RoboDK station: simulator.rdk

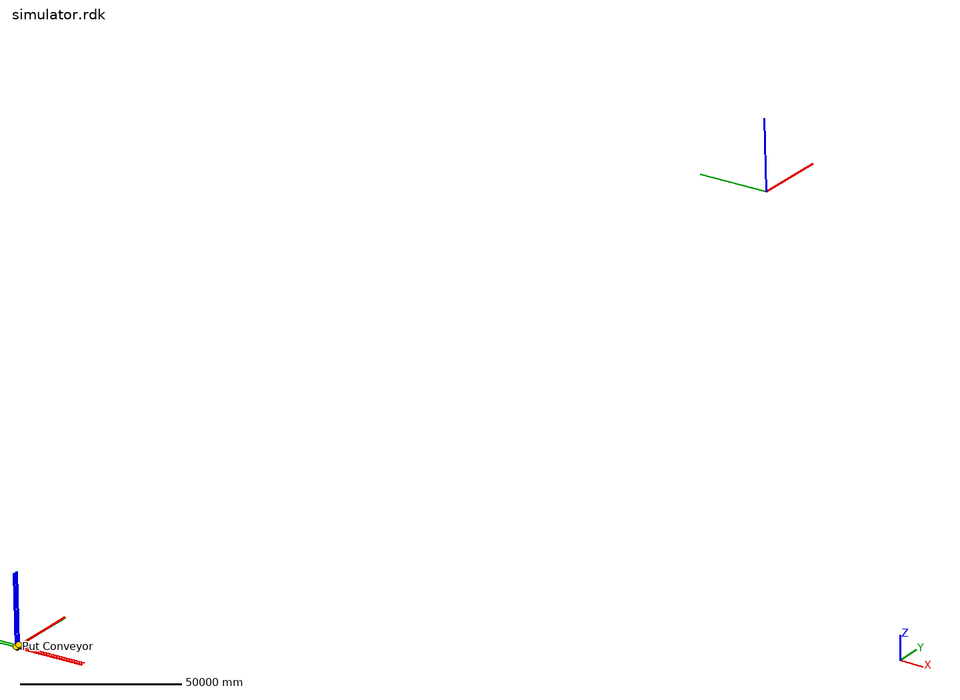
[picture v0: the station drawn from its stored meshes, robots at their saved joint values, targets as dots, program paths as lines]
Station 컨베이어시뮬레이션 (saved by RoboDK 5.8.0). Poses are relative to the parent item; angles as X-Y-Z fixed-axis rotations.
Station parameters (name, value as stored): SizeBox, 50, 50, 50, SizePallet, 2,2,2, ConvSpeed, 50.0, SENSOR, 0
  - frame ConveyorReference at (546.99, -679.94, 19.36) mm, rotated rx -0.64 ry -2.2 rz 0 deg
    - robot Conveyor Belt: 1 axes
        modified DH rows (alpha deg, a mm, theta deg, d mm): 0, 0, 0, 0 linear
        base shift (440, 200, 0) mm, rotated rx 0 ry 90 rz 90 deg
        joint limits [-500000] to [500000]; home [0]; saved at [403823.116]
      - frame MovingRef at (0, 0, 0) mm
        - object box100mm at (-288503.23, 164.8, -52.99) mm, rotated rx 0 ry 0 rz 21.63 deg, size 100 x 100 x 100 mm, geometry from box.sld
        - object Part 4 at (-402571.71, 262.16, 22.01) mm, rotated rx 0 ry 0 rz 28.41 deg, size 50 x 50 x 50 mm, geometry from box.sld
        - object Part 3 at (-402727.14, 262.16, 22.01) mm, rotated rx 0 ry 0 rz 28.12 deg, size 50 x 50 x 50 mm, geometry from box.sld
        - object Part 2 at (-402880.9, 262.16, 22.01) mm, rotated rx 0 ry 0 rz -35.23 deg, size 50 x 50 x 50 mm, geometry from box.sld
        - object Part 1 at (-403045.44, 262.16, 22.01) mm, rotated rx 0 ry 0 rz 36.59 deg, size 50 x 50 x 50 mm, geometry from box.sld
    - target ConveyorHome (joint target) at (440, 200, 0) mm, rotated rx 0 ry 0 rz 90 deg; joints [0] of Conveyor Belt
    - target ConveyorMove (joint target) at (440, 500200, 0) mm, rotated rx 0 ry 0 rz 90 deg; joints [500000] of Conveyor Belt
    - target Put Conveyor (Cartesian target) at (177.84, 575.36, -2.99) mm, rotated rx -180 ry 0 rz 90 deg; joints [-0.131, 70.841, 51.659, -0.131] of UR10 A
    - target Get Conveyor (Cartesian target) at (183.64, 1630.4, -24.46) mm, rotated rx -180 ry 0 rz 90 deg; joints [-9.075, 81.465, 49.928, -9.075] of UR10 B
  - Python program SetSimulationParams (listed below)
  - Python program PrepareSimulation (listed below)
  - Python program SimulateCamera (listed below)
  - Python program PartsToConveyor (listed below)
  - Python program CameraRecognition (listed below)
  - Python program SocketSimulation (listed below)
  - program MoveConveyor (1 instructions, listed below)
  - program MainSimulation (5 instructions, listed below)
  - frame UR10 Base A at (445.82, -104.09, -0.94) mm, rotated rx -0.64 ry -2.2 rz 0 deg
    - robot UR10 A (model Dobot Magician): 4 axes, payload 0.5 kg, reach 320 mm, repeatability 0.2 mm, weight 4 kg
        joint limits [-90, -0.001, -10, -90] to [90, 85, 95, 90]; home [0, 0, 0, 0]; saved at [-0.009, 33.406, -9.672, 20]
      - tool GripperA, TCP at (0, 0, 30) mm, rotated rx 0 ry 0 rz 90 deg, size 209.9 x 42 x 100 mm, geometry from COMPOUND (2)
      - tool TCP A, TCP at (0, 0, 55) mm, rotated rx 0 ry 0 rz 90 deg
    - frame PalletA at (80, -293.6, 0) mm, rotated rx 0 ry 0 rz 90 deg
      - object Europallet at (0, 0, 0) mm, size 192 x 34.6 x 288 mm, geometry from Europallet.sld
    - target ConvApproachA (joint target) at (280.24, -0.04, 215.39) mm, rotated rx -180 ry 0 rz 90 deg; joints [-0.009, 33.406, -9.672, -0.009] of UR10 A
    - target PalletApproachA (joint target) at (2.78, -256.23, 217.48) mm, rotated rx 177.43 ry 0 rz 90 deg; joints [-89.779, 20.936, 0.649, -89.779] of UR10 A
  - frame UR10 Base B at (446.29, 995.84, -13.14) mm, rotated rx -0.64 ry -2.2 rz 0 deg
    - robot UR10 B (model Dobot Magician): 4 axes, payload 0.5 kg, reach 320 mm, repeatability 0.2 mm, weight 4 kg
        joint limits [-90, -0.001, -10, -90] to [90, 85, 95, 90]; home [0, 0, 0, 0]; saved at [-8.952, 40.043, -8.92, 90]
      - tool GripperB, TCP at (0, 0, 30) mm, rotated rx 0 ry 0 rz 90 deg, size 209.9 x 42 x 100 mm, geometry from COMPOUND (2)
      - frame Camera Reference at (0, -70, 0) mm
        - object SICK VSPP-5F2113 Camera at (0, 0, 0) mm, size 116 x 53 x 38 mm, geometry from camera.sld
      - tool TCP B, TCP at (0, 0, 55) mm, rotated rx 0 ry 0 rz 90 deg
    - frame PalletB at (80, 160, 10) mm, rotated rx 0 ry 0 rz 90 deg
      - object Europallet at (0, 0, 20) mm, size 192 x 34.6 x 288 mm, geometry from Europallet.sld
      - object Part 8 at (23.8, -26.65, 46.46) mm, size 50 x 50 x 50 mm, geometry from box.sld
      - object Part 7 at (108.84, -14.03, 46.46) mm, size 50 x 50 x 50 mm, geometry from box.sld
      - object Part 6 at (37.82, 24.09, 46.46) mm, size 50 x 50 x 50 mm, geometry from box.sld
      - object Part 5 at (79.49, 23.53, 46.46) mm, size 50 x 50 x 50 mm, geometry from box.sld
    - target InspectPartB (joint target) at (289.51, -45.6, 234.14) mm, rotated rx 180 ry 0 rz -180 deg; joints [-8.952, 40.043, -8.92, -8.952] of UR10 B
    - target PalletApproachB (joint target) at (9.31, 201.92, 209.08) mm, rotated rx 180 ry 0 rz -180 deg; joints [87.417, 0.29, -9.698, -2.583] of UR10 B
    - target ConvApproachB (joint target) at (9.31, 201.72, 237.71) mm, rotated rx 180 ry 0 rz -180 deg; joints [87.417, 0.29, -9.698, -2.583] of UR10 B
  - camera Camera 1
  - camera Camera 2
  - camera Camera 3
  - camera Camera 4
  - camera Camera 5
  - camera Camera 6
  - camera Camera 7
  - camera Camera 8
  - camera Camera 9
  - camera Camera 10
  - camera Camera 11
  - camera Camera 12
  - camera Camera 13

--- Python program SetSimulationParams ---
# Type help("robolink") or help("robodk") for more information
# Press F5 to run the script
# Note: you do not need to keep a copy of this file, your python script is saved with the station
from robolink import *    # API to communicate with RoboDK
from robodk import *      # basic matrix operations


PARAM_SIZE_BOX = 'SizeBox'
PARAM_SIZE_PALLET = 'SizePallet'
PARAM_CONV_SPEED_MM = 'ConvSpeed'



RDK = Robolink()

size_box = RDK.getParam(PARAM_SIZE_BOX)
size_pallet = RDK.getParam(PARAM_SIZE_PALLET)
conv_speed = RDK.getParam(PARAM_CONV_SPEED_MM)

# ------------------------------------------------------------
size_box_input = mbox('Enter the size of the box in mm [L,W,H]', entry=size_box)
if size_box_input:
    RDK.setParam(PARAM_SIZE_BOX, size_box_input)
else:
    raise Exception('Operation cancelled by user')

# ------------------------------------------------------------
size_pallet_input = mbox('Enter the size of the pallet', entry=size_pallet)
if size_pallet_input:
    RDK.setParam(PARAM_SIZE_PALLET, size_pallet_input)
else:
    raise Exception('Operation cancelled by user')

# ------------------------------------------------------------
conv_speed_input = mbox('Enter the speed of the conveyor in mm/s', entry=conv_speed)
if conv_speed_input:
    RDK.setParam(PARAM_CONV_SPEED_MM, conv_speed_input)
    conv_speed = float(conv_speed_input)
    conv = RDK.Item('Conveyor Belt', ITEM_TYPE_ROBOT)
    conv.setSpeed(conv_speed)

else:
    raise Exception('Operation cancelled by user')

--- Python program PrepareSimulation ---
# Type help("robolink") or help("robodk") for more information
# Press F5 to run the script
# Note: you do not need to keep a copy of this file, your python script is saved with the station
from robolink import *    # API to communicate with RoboDK
from robodk import *      # basic matrix operations

# Use RoboDK API as RL
RDK = Robolink()

frame_pallet        = RDK.Item('PalletA', ITEM_TYPE_FRAME)

# get variable parameters
SIZE_BOX = RDK.getParam('SizeBox')
SIZE_PALLET = RDK.getParam('SizePallet')
SIZE_BOX_XYZ = [float(x.replace(' ','')) for x in SIZE_BOX.split(',')]
SIZE_PALLET_XYZ = [float(x.replace(' ','')) for x in SIZE_PALLET.split(',')]
SIZE_BOX_Z = SIZE_BOX_XYZ[2] # the height of the boxes is important to take into account when approaching the positions

def box_calc(size_xyz, pallet_xyz):
    """Calculates a list of points to store parts in a pallet"""
    [size_x, size_y, size_z] = size_xyz
    [pallet_x, pallet_y, pallet_z] = pallet_xyz
    xyz_list = []
    for h in range(int(pallet_z)):
        for j in range(int(pallet_y)):
            for i in range(int(pallet_x)):
                xyz_list = xyz_list + [[(i+0.5)*size_x, (j+0.5)*size_y, (h+0.5)*size_z]]
    return xyz_list

def parts_setup(frame, positions, size_xyz):
    """Place a list of parts in a reference frame. The part/reference object must have been previously copied to the clipboard."""
    [size_x, size_y, size_z] = size_xyz
    nparts = len(positions)
    cstep = 1.0/(nparts - 1)
    for i in range(nparts):
        newpart = frame.Paste()
        newpart.Scale([size_x/100, size_y/100, size_z/100]) #scale with respect to the reference object (100mm cube)
        newpart.setName('Part ' + str(i+1)) #set item name
        newpart.setPose(transl(positions[i])) #set item position with respect to parent
        newpart.setVisible(True, False) #make item visible but hide the reference frame
        newpart.Recolor([1-cstep*i, cstep*i, 0.2, 1]) #set RGBA color

def cleanup(objects, startswith="Part "):
    """Deletes all objects where the name starts with "startswith", from the provided list of objects."""
    for item in objects:
        if item.Name().startswith(startswith):
            item.Delete()

# turn off rendering (much faster when setting up the station)
RDK.Render(False)

# cleanup previous simulation (generated parts and tools)
all_objects = RDK.ItemList(ITEM_TYPE_OBJECT, False)
cleanup(all_objects, 'Part ')
all_tools = RDK.ItemList(ITEM_TYPE_TOOL, False)
cleanup(all_tools, 'TCP ')

# copy the reference part
partref = RDK.Item('box100mm')
partref.Copy()

#RL.Set_Simulation_Speed(500);
#RL.Set_Simulation_Mode(1)

# calculate an array of positions to get/store the parts
parts_positions = box_calc(SIZE_BOX_XYZ, SIZE_PALLET_XYZ)

# setup/initialise the parts on the palled
parts_setup(frame_pallet, parts_positions, SIZE_BOX_XYZ)

RDK.Render(True)

--- Python program SimulateCamera ---
# Type help("robolink") or help("robodk") for more information
# Press F5 to run the script
# Note: you do not need to keep a copy of this file, your python script is saved with the station
from robolink import *    # API to communicate with RoboDK
from robodk import *      # basic matrix operations
RDK = Robolink()

# Close any open 2D camera views
RDK.Cam2D_Close()

camref = RDK.Item('Camera Reference',ITEM_TYPE_FRAME)

# set parameters in mm and degrees:
# FOV: Field of view in degrees (atan(0.5*height/distance) of the sensor divided by
# FOCAL_LENGHT: focal lenght in mm
# FAR_LENGHT: maximum working distance (in mm)
# SIZE: size of the sensor in pixels
# BG_COLOR: background color (rgb color or named color: AARRGGBB)
# LIGHT_AMBIENT: ambient color (rgb color or named color: AARRGGBB)
# LIGHT_SPECULAR: specular color (rgb color or named color: AARRGGBB)
# LIGHT_DIFFUSE: diffuse color (rgb color or named color: AARRGGBB)


# FOCAL_LENGHT: 초점거리
# FOV: 렌즈를 통해서 사진기가 이미지를 담을 수 있는 각
#
cam_id = RDK.Cam2D_Add(camref, 'FOCAL_LENGHT=6 FOV=32 FAR_LENGHT=250 SIZE=640x480 BG_COLOR=black')
# cam_id = RDK.Cam2D_Add(camref, 'FOCAL_LENGHT=6 FOV=32 FAR_LENGHT=1000 SIZE=640x480')
# cam_id = RDK.Cam2D_Add(camref, 'FOCAL_LENGHT=6 FOV=32 FAR_LENGHT=1000 SIZE=640x480 BG_COLOR=black LIGHT_AMBIENT=red LIGHT_DIFFUSE=#FF00FF00 LIGHT_SPECULAR=black')
# cam_id = RDK.Cam2D_Add(camref, 'FOCAL_LENGHT=6 FOV=32 FAR_LENGHT=1000 SIZE=640x480 DEPTH')
# cam_id = RDK.Cam2D_Add(camref, 'FOCAL_LENGHT=6 FOV=32 FAR_LENGHT=250 SIZE=640x480 BG_COLOR=black LIGHT_AMBIENT=red LIGHT_DIFFUSE=black LIGHT_SPECULAR=white')


# cam_id = RDK.Cam2D_Add(camref, 'FOCAL_LENGHT=6 FOV=32 FAR_LENGHT=1000 SIZE=640x480 LIGHT_AMBIENT=red')

# cam_id = RDK.Cam2D_Add(camref, 'POPUP')

# RDK.Cam2D_Snapshot(RDK.getParam('PATH_OPENSTATION') + "/sample_image.png", cam_id)

--- Python program PartsToConveyor ---
# Type help("robolink") or help("robodk") for more information
# Press F5 to run the script
# Note: you do not need to keep a copy of this file, your python script is saved with the station
from robolink import *    # API to communicate with RoboDK
from robodk import *      # basic matrix operations
from random import uniform

# Use RoboDK API as RL
RDK = Robolink()

# define default approach distance
APPROACH = 70

# gather robot, tool and reference frames from the station
robot               = RDK.Item('UR10 A', ITEM_TYPE_ROBOT)
tool                = RDK.Item('GripperA', ITEM_TYPE_TOOL)
frame_pallet        = RDK.Item('PalletA', ITEM_TYPE_FRAME)
frame_conv          = RDK.Item('ConveyorReference', ITEM_TYPE_FRAME)
frame_conv_moving   = RDK.Item('MovingRef', ITEM_TYPE_FRAME)

# gather targets
target_pallet_safe = RDK.Item('PalletApproachA', ITEM_TYPE_TARGET)
target_conv_safe = RDK.Item('ConvApproachA', ITEM_TYPE_TARGET)
target_conv = RDK.Item('Put Conveyor', ITEM_TYPE_TARGET)

# get variable parameters
SIZE_BOX = RDK.getParam('SizeBox')
SIZE_PALLET = RDK.getParam('SizePallet')
SIZE_BOX_XYZ = [float(x.replace(' ','')) for x in SIZE_BOX.split(',')]
SIZE_PALLET_XYZ = [float(x.replace(' ','')) for x in SIZE_PALLET.split(',')]
SIZE_BOX_Z = SIZE_BOX_XYZ[2] # the height of the boxes is important to take into account when approaching the positions

def box_calc(size_xyz, pallet_xyz):
    """Calculates a list of points to store parts in a pallet"""
    [size_x, size_y, size_z] = size_xyz
    [pallet_x, pallet_y, pallet_z] = pallet_xyz
    xyz_list = []
    for h in range(int(pallet_z)):
        for j in range(int(pallet_y)):
            for i in range(int(pallet_x)):
                xyz_list = xyz_list + [[(i+0.5)*size_x, (j+0.5)*size_y, (h+0.5)*size_z]]
    return xyz_list

def TCP_On(toolitem):
    """Attaches the closest object to the toolitem Htool pose,
    It will also output appropriate function calls on the generated robot program (call to TCP_On)"""
    toolitem.AttachClosest()
    toolitem.RDK().RunMessage('Set air valve on')
    toolitem.RDK().RunProgram('TCP_On()');

def TCP_Off(toolitem, itemleave=0):
    """Detaches the closest object attached to the toolitem Htool pose,
    It will also output appropriate function calls on the generated robot program (call to TCP_Off)"""
    toolitem.DetachAll(itemleave)
    toolitem.RDK().RunMessage('Set air valve off')
    toolitem.RDK().RunProgram('TCP_Off()');

#RL.Set_Simulation_Speed(500);
#RL.Set_Simulation_Mode(1)

# calculate an array of positions to get/store the parts
parts_positions = box_calc(SIZE_BOX_XYZ, SIZE_PALLET_XYZ)

# Calculate a new TCP that takes into account the size of the part (targets are set to the center of the box)
tool_xyzrpw = tool.PoseTool()*transl(0,0,SIZE_BOX_Z/2)
tool_tcp = robot.AddTool(tool_xyzrpw, 'TCP A')

# ---------------------------------------------------------------------------------
# -------------------------- PROGRAM START ----------------------------------------

robot.setPoseTool(tool_tcp)
nparts = len(parts_positions)
i = nparts-1
while i >= 0:
    # ----------- take a part from the pallet ------
    # get the xyz position of part i
    robot.setPoseFrame(frame_pallet)
    part_position_i = parts_positions[i]
    target_i = transl(part_position_i)*rotx(pi)
    target_i_app = target_i * transl(0,0,-(APPROACH+SIZE_BOX_Z))

    # approach to the pallet
    robot.MoveJ(target_pallet_safe)
    # get the box i
    robot.MoveJ(target_i_app)
    robot.MoveL(target_i)
    TCP_On(tool) # attach the closest part
    robot.MoveL(target_i_app)
    robot.MoveJ(target_pallet_safe)

    # ----------- place the box i on the convegor ------
    # approach to the conveyor
    robot.setPoseFrame(frame_conv)
    target_conv_pose = target_conv.Pose()*transl(0,0,-SIZE_BOX_Z/2)

    target_conv_app = target_conv_pose*transl(0,0,-APPROACH)

    robot.MoveJ(target_conv_safe)
    robot.MoveJ(target_conv_app)

    # Place the part at a random position with respect to the target on the conveyor
    # TX = uniform(-150, 150)
    # RZ = uniform(-90*pi/180, +90*pi/180)
    TX = uniform(-50, 50)
    RZ = uniform(-45*pi/180, +45*pi/180)


    robot.MoveL(target_conv_pose*transl(TX,0,0)*rotz(RZ))
    TCP_Off(tool, frame_conv_moving) # detach an place the object in the moving reference frame of the conveyor
    robot.MoveL(target_conv_app)
    robot.MoveJ(target_conv_safe)

    i = i - 1

--- Python program CameraRecognition ---
# Type help("robolink") or help("robodk") for more information
# Press F5 to run the script
# Note: you do not need to keep a copy of this file, your python script is saved with the station
from robolink import *    # API to communicate with RoboDK
from robodk import *      # basic matrix operations

# Use RoboDK API as RL
RDK = Robolink()

# define default approach distance
APPROACH = 100
SENSOR_VARIABLE = 'SENSOR' # station variable
PART_KEYWORD = 'Part' # parts to look for (camera simulation)

# gather robot, tool and reference frames from the station
robot               = RDK.Item('UR10 B', ITEM_TYPE_ROBOT)
tool                = RDK.Item('GripperB', ITEM_TYPE_TOOL)
frame_pallet        = RDK.Item('PalletB', ITEM_TYPE_FRAME)
frame_conv          = RDK.Item('ConveyorReference', ITEM_TYPE_FRAME)
frame_conv_moving   = RDK.Item('MovingRef', ITEM_TYPE_FRAME)

# gather targets
target_pallet_safe = RDK.Item('PalletApproachB', ITEM_TYPE_TARGET)
target_conv_safe = RDK.Item('ConvApproachB', ITEM_TYPE_TARGET)
target_conv = RDK.Item('Get Conveyor', ITEM_TYPE_TARGET)
target_inspect = RDK.Item('InspectPartB', ITEM_TYPE_TARGET)

# get variable parameters
SIZE_BOX = RDK.getParam('SizeBox')
SIZE_PALLET = RDK.getParam('SizePallet')
SIZE_BOX_XYZ = [float(x.replace(' ','')) for x in SIZE_BOX.split(',')]
SIZE_PALLET_XYZ = [float(x.replace(' ','')) for x in SIZE_PALLET.split(',')]
SIZE_BOX_Z = SIZE_BOX_XYZ[2] # the height of the boxes is important to take into account when approaching the positions

camera_ref_conv = target_conv.PoseAbs()

#----------------- camera simulation
# Get all object names to
all_objects = RDK.ItemList(ITEM_TYPE_OBJECT, True)

# Get object items in a list (faster) and filter by keyword
check_objects = []
for i in range(len(all_objects)):
    if all_objects[i].count(PART_KEYWORD) > 0:
        check_objects.append(RDK.Item(all_objects[i]))

# Make sure that there is at least one part that we are expecting
if len(check_objects) == 0:
    raise Exception('No parts to check for. Name at least one part with the name: %s.' % PICKABLE_OBJECTS_KEYWORD)

# simulates the behavior of the camera (returns TX, TY and RZ)
def WaitPartCamera():
    """Simulate camera detection"""
    if RDK.RunMode() == RUNMODE_SIMULATE:
        # Simulate the camera by waiting for an object to be detected
        while True:
            for part in check_objects:
                # calculate the position of the part with respect to the target
                part_pose = invH(camera_ref_conv) * part.PoseAbs()
                tx,ty,tz,rx,ry,rz = pose_2_xyzrpw(part_pose)
                rz = rz * pi/180.0 # Convert degrees to radians
                if abs(tx) < 150 and ty < 50 and abs(tz) < 150 and (part.Color()[1] > 0.5 and part.Color()[0] < 0.5 and part.Color()[2] <0.5):
                    print('Part detected: TX,TY,TZ=%.1f,%.1f,%.1f' % (tx,ty,rz))
                    print(part.Color())
                    return tx, ty, rz
            pause(0.005)
    else:
        RDK.RunProgram('WaitPartCamera')
    return 0,0,0

#-----------------------------

def box_calc(size_xyz, pallet_xyz):
    """Calculates a list of points to store parts in a pallet"""
    [size_x, size_y, size_z] = size_xyz
    [pallet_x, pallet_y, pallet_z] = pallet_xyz
    xyz_list = []
    for h in range(int(pallet_z)):
        for j in range(int(pallet_y)):
            for i in range(int(pallet_x)):
                xyz_list = xyz_list + [[(i+0.5)*size_x, (j+0.5)*size_y, (h+0.5)*size_z]]
    return xyz_list

def TCP_On(toolitem):
    """Attaches the closest object to the toolitem Htool pose,
    It will also output appropriate function calls on the generated robot program (call to TCP_On)"""
    toolitem.AttachClosest()
    toolitem.RDK().RunMessage('Set air valve on')
    toolitem.RDK().RunProgram('TCP_On()');

def TCP_Off(toolitem, itemleave=0):
    """Detaches the closest object attached to the toolitem Htool pose,
    It will also output appropriate function calls on the generated robot program (call to TCP_Off)"""
    #toolitem.DetachClosest(itemleave)
    toolitem.DetachAll(itemleave)
    toolitem.RDK().RunMessage('Set air valve off')
    toolitem.RDK().RunProgram('TCP_Off()');

# calculate an array of positions to get/store the parts
parts_positions = box_calc(SIZE_BOX_XYZ, SIZE_PALLET_XYZ)

# Calculate a new TCP that takes into account the size of the part (targets are set to the center of the box)
tool_xyzrpw = tool.PoseTool()*transl(0,0,SIZE_BOX_Z/2)
tool_tcp = robot.AddTool(tool_xyzrpw, 'TCP B')

# ---------------------------------------------------------------------------------
# -------------------------- PROGRAM START ----------------------------------------
robot.setPoseTool(tool_tcp)
nparts = len(parts_positions)
i = 0
while i < nparts:
    # ----------- take a part from the convegor ------
    # approach to the conveyor
    robot.setPoseFrame(frame_conv)
    robot.MoveJ(target_inspect)

    #------------------------- camera simulation
    CAM_TX, CAM_TY, CAM_RZ = WaitPartCamera()
    # Adjust position along movement according to conveyor speed
    CAM_TY = CAM_TY - 50
    # Lazy move: the part is symmetrical so there is no need to turn more than +/-90 deg around the Z axis. If so, add as many half turns as required
    if CAM_RZ > pi/2:
        CAM_RZ = CAM_RZ - pi
    elif CAM_RZ < -pi/2:
        CAM_RZ = CAM_RZ + pi
    target_conv_pose = target_conv.Pose()*transl(CAM_TX,CAM_TY,-SIZE_BOX_Z/2)*rotz(CAM_RZ)
    target_conv_app = target_conv_pose*transl(0,0,-APPROACH)
    #-------------------------------------------------

    robot.MoveL(target_conv_pose)
    TCP_On(tool) # detach an place the object in the moving reference frame of the conveyor
    robot.MoveL(target_conv_app)

    if len(tool.Childs()) == 0:
        # Detect invalid pick
        continue

    print(1)
    robot.MoveJ(target_conv_safe)

    # ----------- place the part on the pallet ------
    # get the xyz position of part i
    robot.setPoseFrame(frame_pallet)
    part_position_i = parts_positions[i]
    target_i = transl(part_position_i)*rotx(pi)
    target_i_app = target_i * transl(0,0,0)
    # approach to the pallet
    print(2)
    robot.MoveJ(target_pallet_safe)
    print(3)
    # get the box i
    robot.MoveJ(target_i_app)
    robot.MoveL(target_i)
    TCP_Off(tool, frame_pallet) # attach the closest part
    robot.MoveL(target_i_app)
    robot.MoveJ(target_pallet_safe)

    i = i + 1

--- Python program SocketSimulation ---
from robolink import *
from robodk import *

import_install("websockets")
import asyncio
import websockets
import json

RDK = Robolink()

robotA = RDK.Item("UR10 A")
robotA_joints = robotA.Joints().list()
robotA_x = robotA_joints[0]
robotA_y = robotA_joints[1]
robotA_z = robotA_joints[2]
robotA_rotation = robotA_joints[3]
print(robotA_x, robotA_y, robotA_z, robotA_rotation)
robotB = RDK.Item("UR10 B")
robotB_joints = robotB.Joints().list()
robotB_x = robotB_joints[0]
robotB_y = robotB_joints[1]
robotB_z = robotB_joints[2]
robotB_rotation = robotB_joints[3]

PARAM_CONV_SPEED_MM = 'ConvSpeed'
conv_speed = RDK.getParam(PARAM_CONV_SPEED_MM)
conv = RDK.Item('Conveyor Belt', ITEM_TYPE_ROBOT)

# 각 상황에 따라 URL 을 변경해주세요.
# 실행을 위해 websockets 설치가 필요합니다.
# RoboDK - 도구 - 스크립트 실행 - Install Python Package - websockets

# production
# SERVER_URL = "robots.mincodinglab.com"

# dev
SERVER_URL = "localhost:8000"

async def connect():
    uri = f"ws://{SERVER_URL}/socket/ws/robodk/"
    async with websockets.connect(uri) as websocket:
        RDK.ShowMessage("Connection established!", False)

        while True:
            try:
                # 서버로부터 메시지 수신
                response = await websocket.recv()

                data = json.loads(response)
                message = json.loads(data.get('message'))
                if message.get("robotA_joint1"):
                    robotA.MoveJ([int(message.get("robotA_joint1")), robotA_y, robotA_z, robotA_rotation])
                elif message.get("robotA_joint2"):
                    robotA.MoveJ([robotA_x, int(message.get("robotA_joint2")), robotA_z, robotA_rotation])
                elif message.get("robotA_joint3"):
                    robotA.MoveJ([robotA_x, robotA_y, int(message.get("robotA_joint3")), robotA_rotation])
                elif message.get("robotA_joint4"):
                    robotA.MoveJ([robotA_x, robotA_y, robotA_z, int(message.get("robotA_joint4"))])
                elif message.get("robotB_joint1"):
                    robotB.MoveJ([int(message.get("robotB_joint1")), robotB_y, robotB_z, robotB_rotation])
                elif message.get("robotB_joint2"):
                    robotB.MoveJ([robotB_x, int(message.get("robotB_joint2")), robotB_z, robotB_rotation])
                elif message.get("robotB_joint3"):
                    robotB.MoveJ([robotB_x, robotB_y, int(message.get("robotB_joint3")), robotB_rotation])
                elif message.get("robotB_joint4"):
                    robotB.MoveJ([robotB_x, robotB_y, robotB_z, int(message.get("robotB_joint4"))])
                elif message.get("program"):
                    flag = message.get("program")
                    if flag == "start":
                        RDK.RunCode("PrepareSimulation")
                        pause(1)
                        RDK.RunCode("MoveConveyor")
                        RDK.RunCode("SimulateCamera")
                        pause(1)
                        RDK.RunCode("CameraRecognition")
                        RDK.RunCode("PartsToConveyor")
                    elif flag == "stop":
                        programs = RDK.ItemList(ITEM_TYPE_PROGRAM)
                        for prog in programs:
                            prog.Stop()

                        programs = RDK.ItemList(ITEM_TYPE_PROGRAM_PYTHON)
                        for prog in programs:
                            prog.Stop()



            except websockets.ConnectionClosed:
                RDK.ShowMessage("Connection closed", False)
                break
            except Exception as e:
                RDK.ShowMessage(f"WebSocket Error: {e}", False)
                break

async def main():
    await connect()

if __name__ == "__main__":
    asyncio.run(main())

--- program MoveConveyor (robot Conveyor Belt) ---
  MoveJ (ConveyorMove)

--- program MainSimulation ---
  Call PrepareSimulation
  Run MoveConveyor
  Call SimulateCamera
  Run CameraRecognition
  Call PartsToConveyor
